(* Logix 5000 project; controller PROJECT2 Emulate 5570 rev 30.12; software revision 30.01; part 3 of 3 *)
(* tags used below, declared in another part *)
   BottleCapped : COUNTER;
   BottleFilled : COUNTER;
   BottlePresentAt4 : TIMER;
   BottlePresentTimer : TIMER;
   CapInsertTimer : TIMER;
   CurrentHeightFilled : DINT;
   CycleTimer : TIMER;
   CycleTimer2 : TIMER;
   Filled : COUNTER;
   filler : BOOL;
   FillerDownTMR : TIMER;
   FillerFilledTMR : TIMER;
   HeightFilled : DINT;
   HEIGHTFILLEDONESHOT : BOOL;
   In : DINT;
   OutPutOneShot : BOOL;
   SIM_BNOP : BOOL;
   SIM_LevelSensor : AOI_SIMAnalogSensor_OnOff;
   SIM_ONS : BOOL;
   SIM_OutfeedSensor : AOI_SIMPartSensor;
   SIM_PowerONPB : BOOL;
   SIM_PPENABLED : BOOL;
   SIM_PTInfeedToStn1 : AOI_SIMPartTravel;
   SIM_PTStn2Fill : AOI_SIMPartTravel;
   SIM_PTStn4ToOutfeed : AOI_SIMPartTravel;
   SIM_PTStnStatus : StationStatus[20];
   SIM_PTWalkingBeam : AOI_SIMPartTravel;
   SIM_SpeedSensor : AOI_SIMAnalogSensor_OnOff;
   SIM_Stn1BottlePresentSensor : AOI_SIMPartSensor;
   SIM_Stn2BottleFilledSensor : AOI_SIMPartSensor;
   SIM_Stn2BottlePresentSensor : AOI_SIMPartSensor;
   SIM_Stn2Filler_Cylinder : AOI_SIM_2PosCyl_RsLwr;
   SIM_Stn2Filler_Fill : AOI_SIM_SimpleValve;
   SIM_Stn3BottlePresentSensor : AOI_SIMPartSensor;
   SIM_Stn3CapInsert : AOI_SIM_2PosCyl_RsLwr;
   SIM_Stn3CapPresentSensor : AOI_SIMPartSensor;
   SIM_Stn4BottlePresentSensor : AOI_SIMPartSensor;
   SIM_Stn4CapRotate : AOI_SIM_Conveyor;
   SIM_Stn4CapRotate_Cylinder : AOI_SIM_2PosCyl_RsLwr;
   SIM_WalkingBeam : AOI_SIM_3PosCyl_ExtRet;
   SIM_WalkingBeamClamp : AOI_SIM_2PosCyl_ExtRet;
   SIM_Zero : DINT;
   St4CycleTime : TIMER;
   station2oneshot : BOOL;
   Station3OneShot : BOOL;
   Station4OneShot : BOOL;
   Station4OneShot2 : BOOL;
   Station4OneShot3 : BOOL;
   TotalCycleTime : REAL;
   TotalFilledHEight : DINT;
   CH0 : ALIAS FOR Local:4:I.Ch0Data;
   CH1 : ALIAS FOR Local:4:I.Ch1Data;
   I2 : ALIAS FOR Local:2:I.Data;
   I31 : ALIAS FOR Ethernet3_PointIO:1:I;
   I32 : ALIAS FOR Ethernet3_PointIO:2:I;
   I33 : ALIAS FOR Ethernet3_PointIO:3:I;
   O3 : ALIAS FOR Local:3:O.Data;
   O34 : ALIAS FOR Ethernet3_PointIO:4:O;
   O35 : ALIAS FOR Ethernet3_PointIO:5:O;
   O36 : ALIAS FOR Ethernet3_PointIO:6:O;
   TP : TouchPanel;
(* MainProgram, continued *)

ROUTINE Filling_R02   (* ladder *)
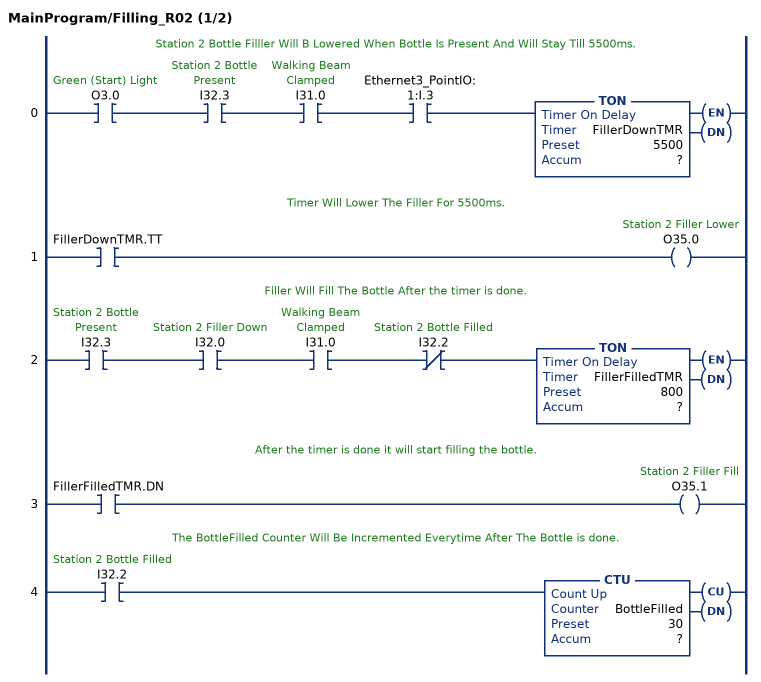
   // Station 2 Bottle Filller Will B Lowered When Bottle Is Present And Will Stay Till 5500ms.
   0: XIC(O3.0)XIC(I32.3)XIC(I31.0)XIC(Ethernet3_PointIO:1:I.3)TON(FillerDownTMR,?,?);
   // Timer Will Lower The Filler For 5500ms.
   1: XIC(FillerDownTMR.TT)OTE(O35.0);
   // Filler Will Fill The Bottle After the timer is done.
   2: XIC(I32.3)XIC(I32.0)XIC(I31.0)XIO(I32.2)TON(FillerFilledTMR,?,?);
   // After the timer is done it will start filling the bottle.
   3: XIC(FillerFilledTMR.DN)OTE(O35.1);
   // The BottleFilled Counter Will Be Incremented Everytime After The Bottle is done.
   4: XIC(I32.2)CTU(BottleFilled,?,?);
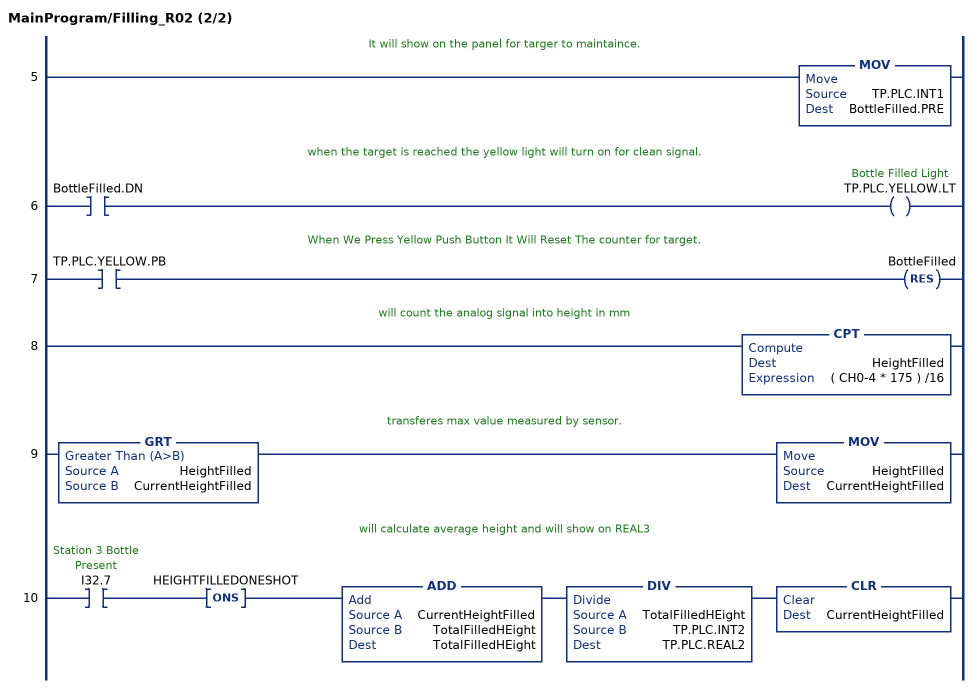
   // It will show on the panel for targer to maintaince.
   5: MOV(TP.PLC.INT1,BottleFilled.PRE);
   // when the target is reached the yellow light will turn on for clean signal.
   6: XIC(BottleFilled.DN)OTE(TP.PLC.YELLOW.LT);
   // When We Press Yellow Push Button It Will Reset The counter for target.
   7: XIC(TP.PLC.YELLOW.PB)RES(BottleFilled);
   // will count the analog signal into height in mm
   8: CPT(HeightFilled,( CH0-4 * 175 ) /16);
   // transferes max value measured by sensor.
   9: GRT(HeightFilled,CurrentHeightFilled)MOV(HeightFilled,CurrentHeightFilled);
   // will calculate average height and will show on REAL3
   10: XIC(I32.7)ONS(HEIGHTFILLEDONESHOT)ADD(CurrentHeightFilled,TotalFilledHEight,TotalFilledHEight)DIV(TotalFilledHEight,TP.PLC.INT2,TP.PLC.REAL2)CLR(CurrentHeightFilled);
END_ROUTINE

ROUTINE MainRoutine   (* ladder *)
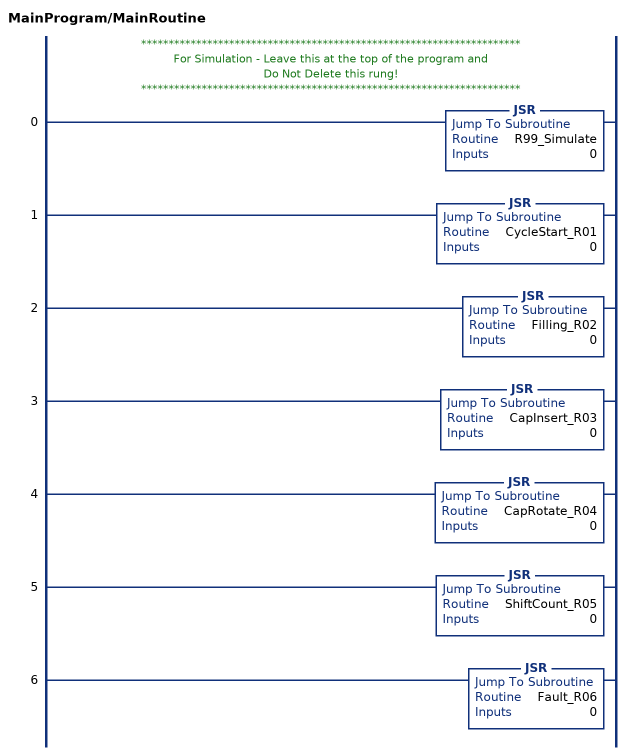
   // *********************************************************************
   // For Simulation - Leave this at the top of the program and
   // Do Not Delete this rung!
   // *********************************************************************
   0: JSR(R99_Simulate,0);
   1: JSR(CycleStart_R01,0);
   2: JSR(Filling_R02,0);
   3: JSR(CapInsert_R03,0);
   4: JSR(CapRotate_R04,0);
   5: JSR(ShiftCount_R05,0);
   6: JSR(Fault_R06,0);
END_ROUTINE

ROUTINE R99_Simulate   (* ladder *)
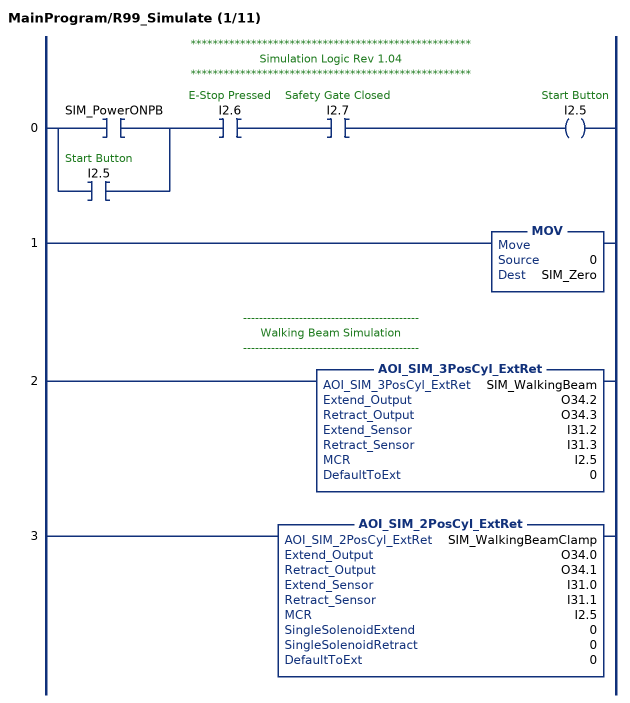
   // ***************************************************
   // Simulation Logic Rev 1.04
   // ***************************************************
   0: [XIC(SIM_PowerONPB) ,XIC(I2.5) ]XIC(I2.6)XIC(I2.7)OTE(I2.5);
   1: MOV(0,SIM_Zero);
   // --------------------------------------------
   // Walking Beam Simulation
   // --------------------------------------------
   2: AOI_SIM_3PosCyl_ExtRet(SIM_WalkingBeam,O34.2,O34.3,I31.2,I31.3,I2.5,0);
   3: AOI_SIM_2PosCyl_ExtRet(SIM_WalkingBeamClamp,O34.0,O34.1,I31.0,I31.1,I2.5,0,0,0);
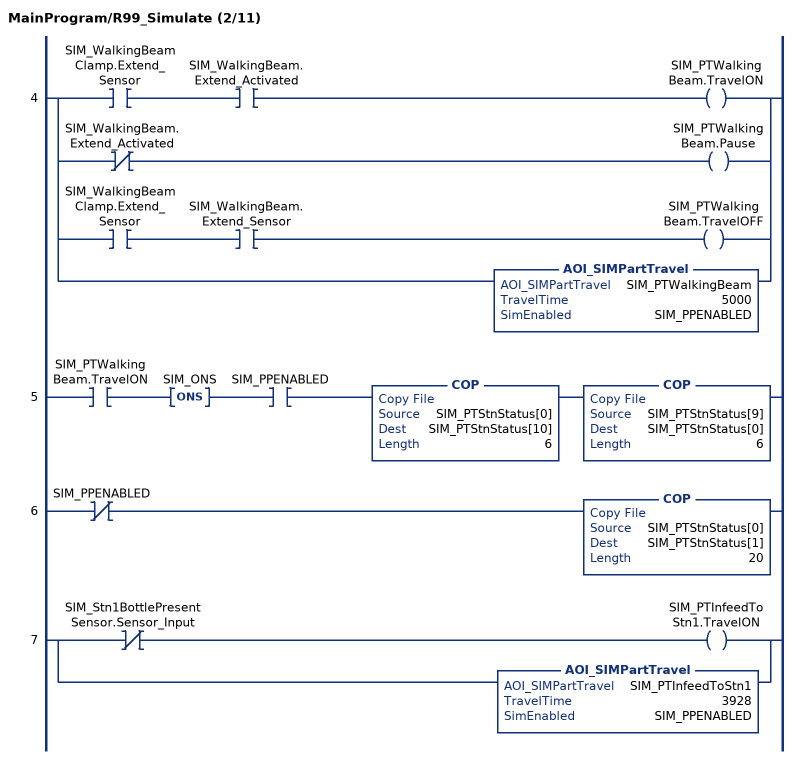
   4: [XIC(SIM_WalkingBeamClamp.Extend_Sensor) XIC(SIM_WalkingBeam.Extend_Activated) OTE(SIM_PTWalkingBeam.TravelON) ,XIO(SIM_WalkingBeam.Extend_Activated) OTE(SIM_PTWalkingBeam.Pause) ,XIC(SIM_WalkingBeamClamp.Extend_Sensor) XIC(SIM_WalkingBeam.Extend_Sensor) OTE(SIM_PTWalkingBeam.TravelOFF) ,AOI_SIMPartTravel(SIM_PTWalkingBeam,5000,SIM_PPENABLED) ];
   5: XIC(SIM_PTWalkingBeam.TravelON)ONS(SIM_ONS)XIC(SIM_PPENABLED)COP(SIM_PTStnStatus[0],SIM_PTStnStatus[10],6)COP(SIM_PTStnStatus[9],SIM_PTStnStatus[0],6);
   6: XIO(SIM_PPENABLED)COP(SIM_PTStnStatus[0],SIM_PTStnStatus[1],20);
   7: [XIO(SIM_Stn1BottlePresentSensor.Sensor_Input) OTE(SIM_PTInfeedToStn1.TravelON) ,AOI_SIMPartTravel(SIM_PTInfeedToStn1,3928,SIM_PPENABLED) ];
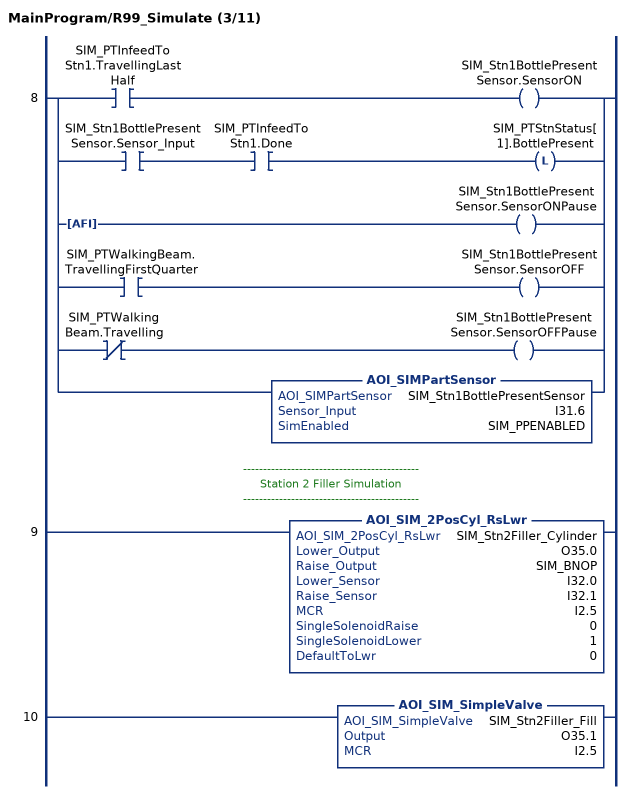
   8: [XIC(SIM_PTInfeedToStn1.TravellingLastHalf) OTE(SIM_Stn1BottlePresentSensor.SensorON) ,XIC(SIM_Stn1BottlePresentSensor.Sensor_Input) XIC(SIM_PTInfeedToStn1.Done) OTL(SIM_PTStnStatus[1].BottlePresent) ,AFI() OTE(SIM_Stn1BottlePresentSensor.SensorONPause) ,XIC(SIM_PTWalkingBeam.TravellingFirstQuarter) OTE(SIM_Stn1BottlePresentSensor.SensorOFF) ,XIO(SIM_PTWalkingBeam.Travelling) OTE(SIM_Stn1BottlePresentSensor.SensorOFFPause) ,AOI_SIMPartSensor(SIM_Stn1BottlePresentSensor,I31.6,SIM_PPENABLED) ];
   // --------------------------------------------
   // Station 2 Filler Simulation
   // --------------------------------------------
   9: AOI_SIM_2PosCyl_RsLwr(SIM_Stn2Filler_Cylinder,O35.0,SIM_BNOP,I32.0,I32.1,I2.5,0,1,0);
   10: AOI_SIM_SimpleValve(SIM_Stn2Filler_Fill,O35.1,I2.5);
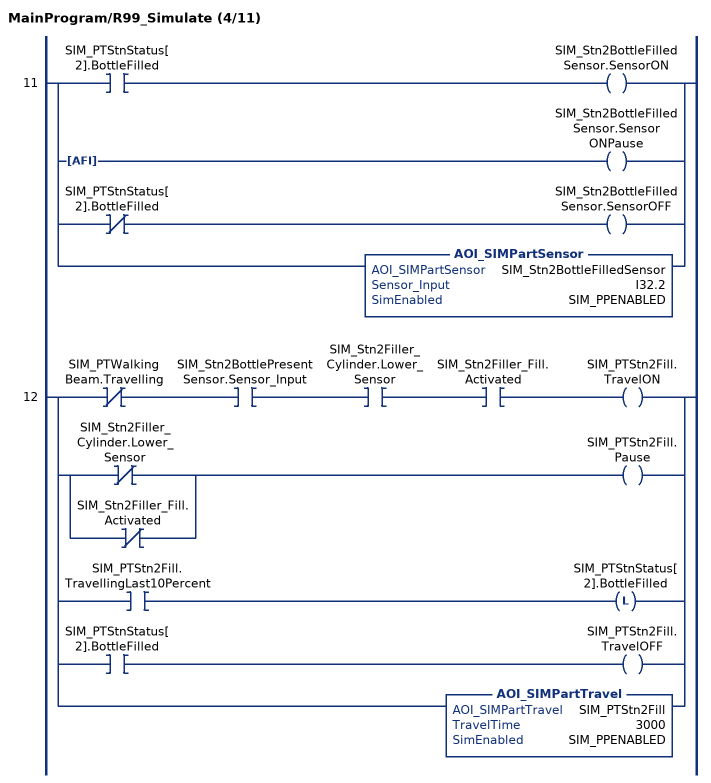
   11: [XIC(SIM_PTStnStatus[2].BottleFilled) OTE(SIM_Stn2BottleFilledSensor.SensorON) ,AFI() OTE(SIM_Stn2BottleFilledSensor.SensorONPause) ,XIO(SIM_PTStnStatus[2].BottleFilled) OTE(SIM_Stn2BottleFilledSensor.SensorOFF) ,AOI_SIMPartSensor(SIM_Stn2BottleFilledSensor,I32.2,SIM_PPENABLED) ];
   12: [XIO(SIM_PTWalkingBeam.Travelling) XIC(SIM_Stn2BottlePresentSensor.Sensor_Input) XIC(SIM_Stn2Filler_Cylinder.Lower_Sensor) XIC(SIM_Stn2Filler_Fill.Activated) OTE(SIM_PTStn2Fill.TravelON) ,[XIO(SIM_Stn2Filler_Cylinder.Lower_Sensor) ,XIO(SIM_Stn2Filler_Fill.Activated) ] OTE(SIM_PTStn2Fill.Pause) ,XIC(SIM_PTStn2Fill.TravellingLast10Percent) OTL(SIM_PTStnStatus[2].BottleFilled) ,XIC(SIM_PTStnStatus[2].BottleFilled) OTE(SIM_PTStn2Fill.TravelOFF) ,AOI_SIMPartTravel(SIM_PTStn2Fill,3000,SIM_PPENABLED) ];
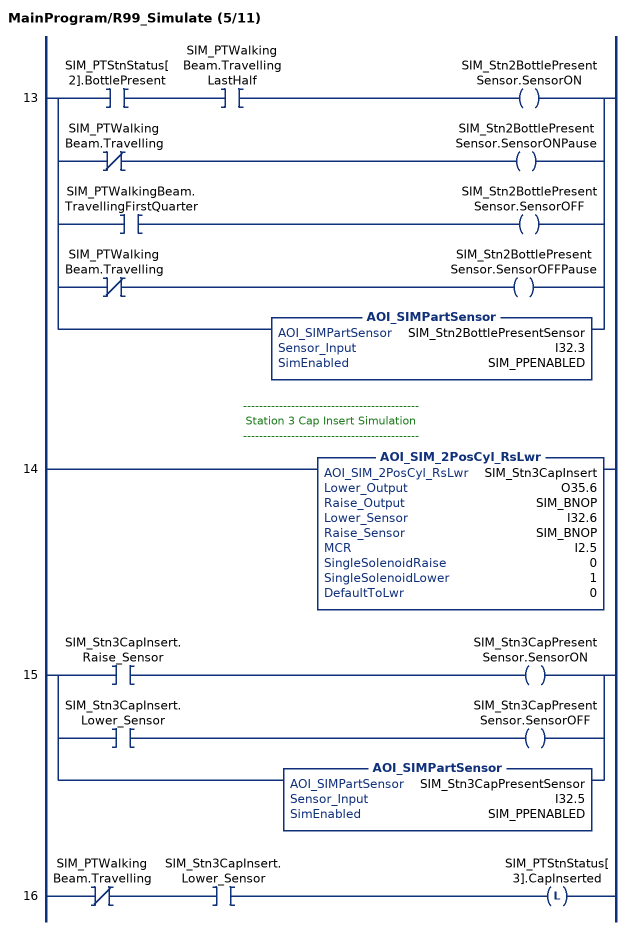
   13: [XIC(SIM_PTStnStatus[2].BottlePresent) XIC(SIM_PTWalkingBeam.TravellingLastHalf) OTE(SIM_Stn2BottlePresentSensor.SensorON) ,XIO(SIM_PTWalkingBeam.Travelling) OTE(SIM_Stn2BottlePresentSensor.SensorONPause) ,XIC(SIM_PTWalkingBeam.TravellingFirstQuarter) OTE(SIM_Stn2BottlePresentSensor.SensorOFF) ,XIO(SIM_PTWalkingBeam.Travelling) OTE(SIM_Stn2BottlePresentSensor.SensorOFFPause) ,AOI_SIMPartSensor(SIM_Stn2BottlePresentSensor,I32.3,SIM_PPENABLED) ];
   // --------------------------------------------
   // Station 3 Cap Insert Simulation
   // --------------------------------------------
   14: AOI_SIM_2PosCyl_RsLwr(SIM_Stn3CapInsert,O35.6,SIM_BNOP,I32.6,SIM_BNOP,I2.5,0,1,0);
   15: [XIC(SIM_Stn3CapInsert.Raise_Sensor) OTE(SIM_Stn3CapPresentSensor.SensorON) ,XIC(SIM_Stn3CapInsert.Lower_Sensor) OTE(SIM_Stn3CapPresentSensor.SensorOFF) ,AOI_SIMPartSensor(SIM_Stn3CapPresentSensor,I32.5,SIM_PPENABLED) ];
   16: XIO(SIM_PTWalkingBeam.Travelling)XIC(SIM_Stn3CapInsert.Lower_Sensor)OTL(SIM_PTStnStatus[3].CapInserted);
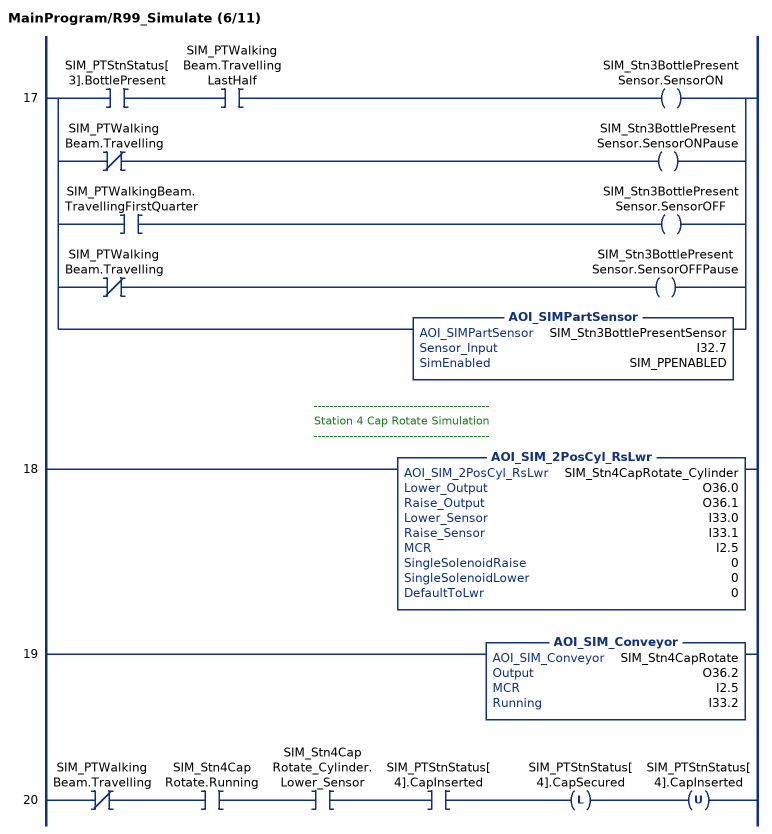
   17: [XIC(SIM_PTStnStatus[3].BottlePresent) XIC(SIM_PTWalkingBeam.TravellingLastHalf) OTE(SIM_Stn3BottlePresentSensor.SensorON) ,XIO(SIM_PTWalkingBeam.Travelling) OTE(SIM_Stn3BottlePresentSensor.SensorONPause) ,XIC(SIM_PTWalkingBeam.TravellingFirstQuarter) OTE(SIM_Stn3BottlePresentSensor.SensorOFF) ,XIO(SIM_PTWalkingBeam.Travelling) OTE(SIM_Stn3BottlePresentSensor.SensorOFFPause) ,AOI_SIMPartSensor(SIM_Stn3BottlePresentSensor,I32.7,SIM_PPENABLED) ];
   // --------------------------------------------
   // Station 4 Cap Rotate Simulation
   // --------------------------------------------
   18: AOI_SIM_2PosCyl_RsLwr(SIM_Stn4CapRotate_Cylinder,O36.0,O36.1,I33.0,I33.1,I2.5,0,0,0);
   19: AOI_SIM_Conveyor(SIM_Stn4CapRotate,O36.2,I2.5,I33.2);
   20: XIO(SIM_PTWalkingBeam.Travelling)XIC(SIM_Stn4CapRotate.Running)XIC(SIM_Stn4CapRotate_Cylinder.Lower_Sensor)XIC(SIM_PTStnStatus[4].CapInserted)OTL(SIM_PTStnStatus[4].CapSecured)OTU(SIM_PTStnStatus[4].CapInserted);
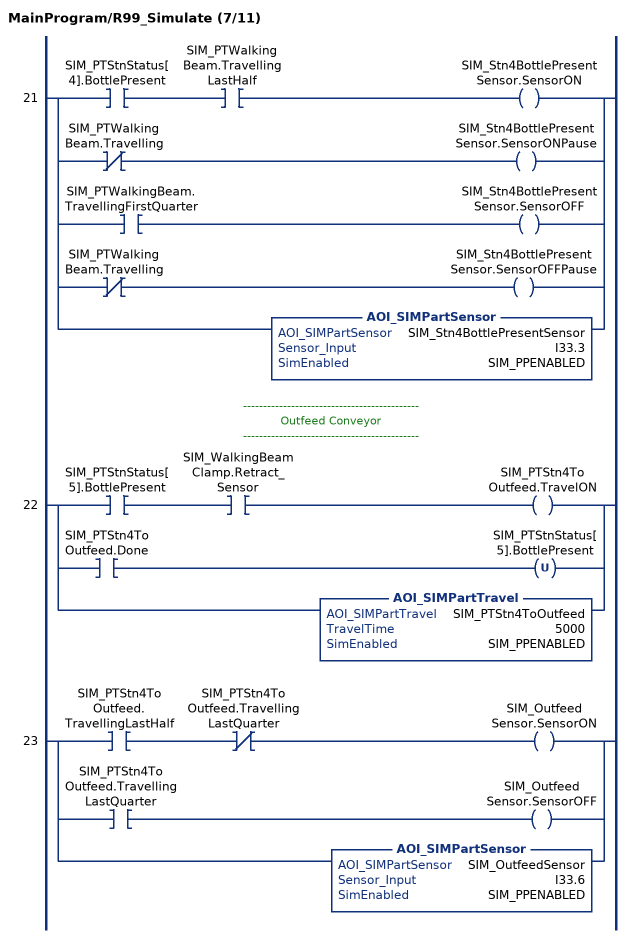
   21: [XIC(SIM_PTStnStatus[4].BottlePresent) XIC(SIM_PTWalkingBeam.TravellingLastHalf) OTE(SIM_Stn4BottlePresentSensor.SensorON) ,XIO(SIM_PTWalkingBeam.Travelling) OTE(SIM_Stn4BottlePresentSensor.SensorONPause) ,XIC(SIM_PTWalkingBeam.TravellingFirstQuarter) OTE(SIM_Stn4BottlePresentSensor.SensorOFF) ,XIO(SIM_PTWalkingBeam.Travelling) OTE(SIM_Stn4BottlePresentSensor.SensorOFFPause) ,AOI_SIMPartSensor(SIM_Stn4BottlePresentSensor,I33.3,SIM_PPENABLED) ];
   // --------------------------------------------
   // Outfeed Conveyor
   // --------------------------------------------
   22: [XIC(SIM_PTStnStatus[5].BottlePresent) XIC(SIM_WalkingBeamClamp.Retract_Sensor) OTE(SIM_PTStn4ToOutfeed.TravelON) ,XIC(SIM_PTStn4ToOutfeed.Done) OTU(SIM_PTStnStatus[5].BottlePresent) ,AOI_SIMPartTravel(SIM_PTStn4ToOutfeed,5000,SIM_PPENABLED) ];
   23: [XIC(SIM_PTStn4ToOutfeed.TravellingLastHalf) XIO(SIM_PTStn4ToOutfeed.TravellingLastQuarter) OTE(SIM_OutfeedSensor.SensorON) ,XIC(SIM_PTStn4ToOutfeed.TravellingLastQuarter) OTE(SIM_OutfeedSensor.SensorOFF) ,AOI_SIMPartSensor(SIM_OutfeedSensor,I33.6,SIM_PPENABLED) ];
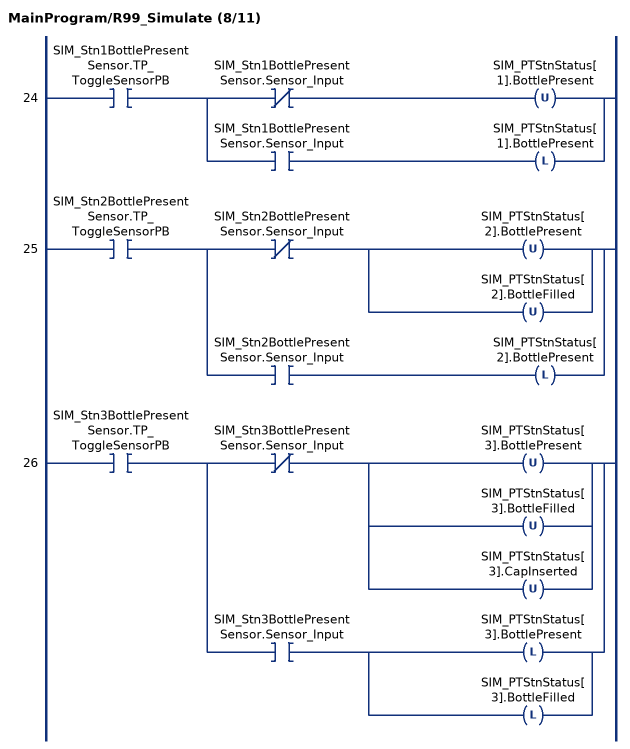
   24: XIC(SIM_Stn1BottlePresentSensor.TP_ToggleSensorPB)[XIO(SIM_Stn1BottlePresentSensor.Sensor_Input) OTU(SIM_PTStnStatus[1].BottlePresent) ,XIC(SIM_Stn1BottlePresentSensor.Sensor_Input) OTL(SIM_PTStnStatus[1].BottlePresent) ];
   25: XIC(SIM_Stn2BottlePresentSensor.TP_ToggleSensorPB)[XIO(SIM_Stn2BottlePresentSensor.Sensor_Input) [OTU(SIM_PTStnStatus[2].BottlePresent) ,OTU(SIM_PTStnStatus[2].BottleFilled) ] ,XIC(SIM_Stn2BottlePresentSensor.Sensor_Input) OTL(SIM_PTStnStatus[2].BottlePresent) ];
   26: XIC(SIM_Stn3BottlePresentSensor.TP_ToggleSensorPB)[XIO(SIM_Stn3BottlePresentSensor.Sensor_Input) [OTU(SIM_PTStnStatus[3].BottlePresent) ,OTU(SIM_PTStnStatus[3].BottleFilled) ,OTU(SIM_PTStnStatus[3].CapInserted) ] ,XIC(SIM_Stn3BottlePresentSensor.Sensor_Input) [OTL(SIM_PTStnStatus[3].BottlePresent) ,OTL(SIM_PTStnStatus[3].BottleFilled) ] ];
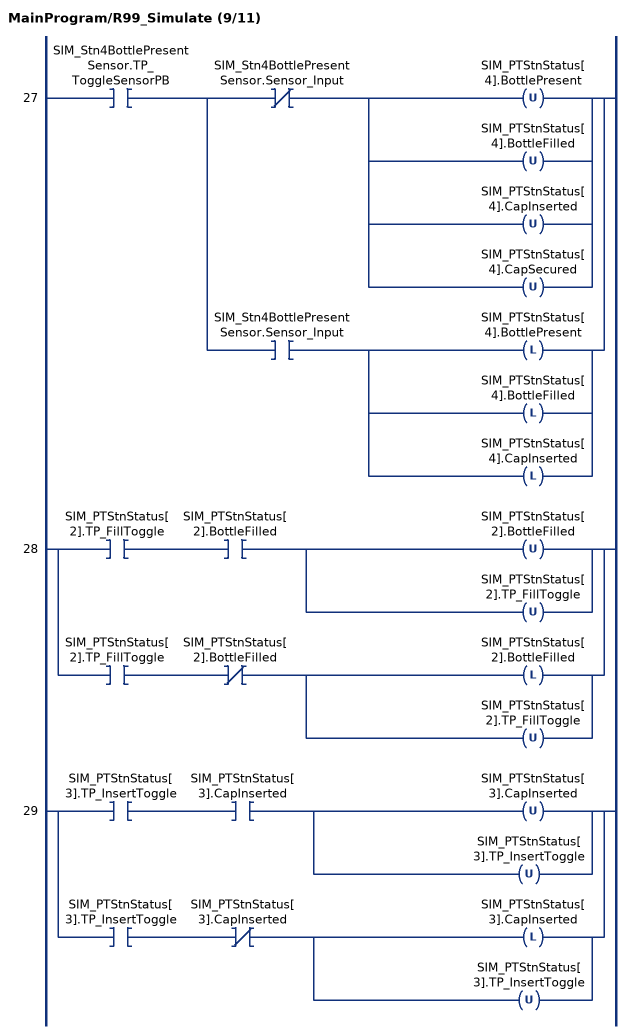
   27: XIC(SIM_Stn4BottlePresentSensor.TP_ToggleSensorPB)[XIO(SIM_Stn4BottlePresentSensor.Sensor_Input) [OTU(SIM_PTStnStatus[4].BottlePresent) ,OTU(SIM_PTStnStatus[4].BottleFilled) ,OTU(SIM_PTStnStatus[4].CapInserted) ,OTU(SIM_PTStnStatus[4].CapSecured) ] ,XIC(SIM_Stn4BottlePresentSensor.Sensor_Input) [OTL(SIM_PTStnStatus[4].BottlePresent) ,OTL(SIM_PTStnStatus[4].BottleFilled) ,OTL(SIM_PTStnStatus[4].CapInserted) ] ];
   28: [XIC(SIM_PTStnStatus[2].TP_FillToggle) XIC(SIM_PTStnStatus[2].BottleFilled) [OTU(SIM_PTStnStatus[2].BottleFilled) ,OTU(SIM_PTStnStatus[2].TP_FillToggle) ] ,XIC(SIM_PTStnStatus[2].TP_FillToggle) XIO(SIM_PTStnStatus[2].BottleFilled) [OTL(SIM_PTStnStatus[2].BottleFilled) ,OTU(SIM_PTStnStatus[2].TP_FillToggle) ] ];
   29: [XIC(SIM_PTStnStatus[3].TP_InsertToggle) XIC(SIM_PTStnStatus[3].CapInserted) [OTU(SIM_PTStnStatus[3].CapInserted) ,OTU(SIM_PTStnStatus[3].TP_InsertToggle) ] ,XIC(SIM_PTStnStatus[3].TP_InsertToggle) XIO(SIM_PTStnStatus[3].CapInserted) [OTL(SIM_PTStnStatus[3].CapInserted) ,OTU(SIM_PTStnStatus[3].TP_InsertToggle) ] ];
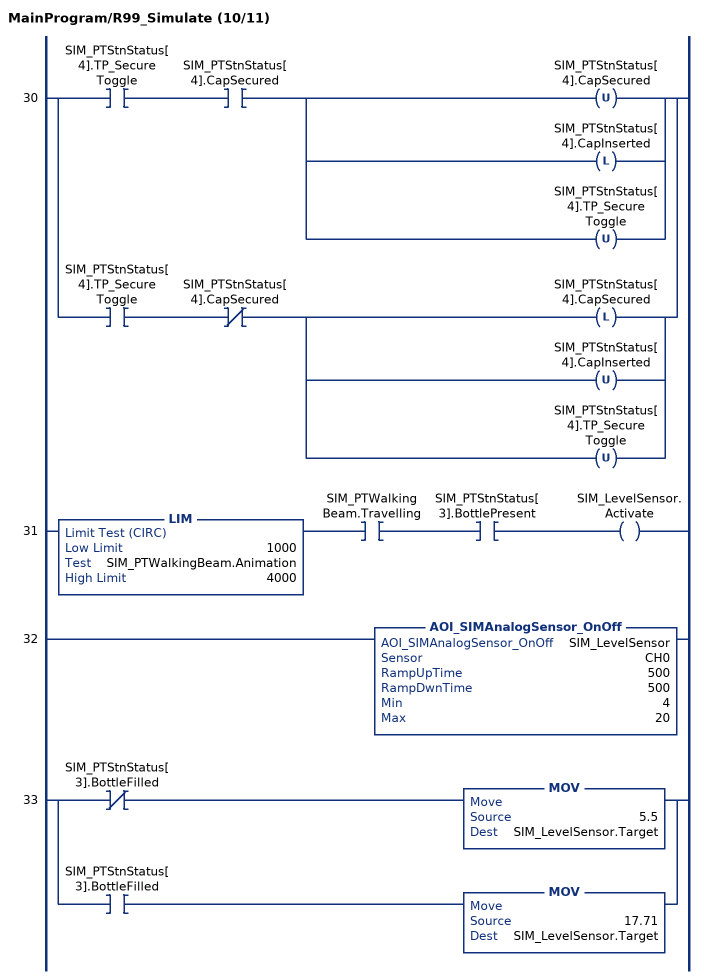
   30: [XIC(SIM_PTStnStatus[4].TP_SecureToggle) XIC(SIM_PTStnStatus[4].CapSecured) [OTU(SIM_PTStnStatus[4].CapSecured) ,OTL(SIM_PTStnStatus[4].CapInserted) ,OTU(SIM_PTStnStatus[4].TP_SecureToggle) ] ,XIC(SIM_PTStnStatus[4].TP_SecureToggle) XIO(SIM_PTStnStatus[4].CapSecured) [OTL(SIM_PTStnStatus[4].CapSecured) ,OTU(SIM_PTStnStatus[4].CapInserted) ,OTU(SIM_PTStnStatus[4].TP_SecureToggle) ] ];
   31: LIM(1000,SIM_PTWalkingBeam.Animation,4000)XIC(SIM_PTWalkingBeam.Travelling)XIC(SIM_PTStnStatus[3].BottlePresent)OTE(SIM_LevelSensor.Activate);
   32: AOI_SIMAnalogSensor_OnOff(SIM_LevelSensor,CH0,500,500,4,20);
   33: [XIO(SIM_PTStnStatus[3].BottleFilled) MOV(5.5,SIM_LevelSensor.Target) ,XIC(SIM_PTStnStatus[3].BottleFilled) MOV(17.71,SIM_LevelSensor.Target) ];
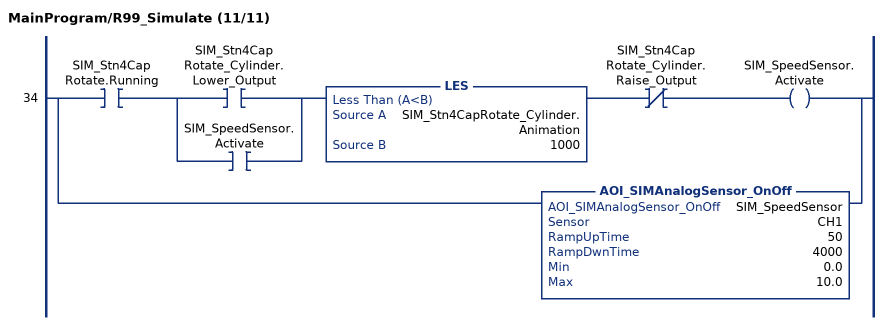
   34: [XIC(SIM_Stn4CapRotate.Running) [XIC(SIM_Stn4CapRotate_Cylinder.Lower_Output) ,XIC(SIM_SpeedSensor.Activate) ] LES(SIM_Stn4CapRotate_Cylinder.Animation,1000) XIO(SIM_Stn4CapRotate_Cylinder.Raise_Output) OTE(SIM_SpeedSensor.Activate) ,AOI_SIMAnalogSensor_OnOff(SIM_SpeedSensor,CH1,50,4000,0.0,10.0) ];
END_ROUTINE

ROUTINE ShiftCount_R05   (* ladder *)
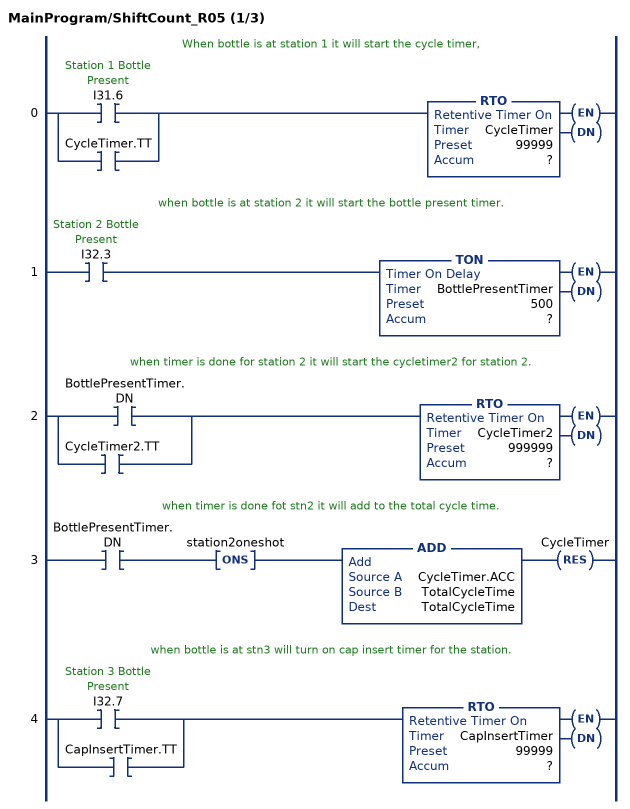
   // When bottle is at station 1 it will start the cycle timer,
   0: [XIC(I31.6) ,XIC(CycleTimer.TT) ]RTO(CycleTimer,?,?);
   // when bottle is at station 2 it will start the bottle present timer.
   1: XIC(I32.3)TON(BottlePresentTimer,?,?);
   // when timer is done for station 2 it will start the cycletimer2 for station 2.
   2: [XIC(BottlePresentTimer.DN) ,XIC(CycleTimer2.TT) ]RTO(CycleTimer2,?,?);
   // when timer is done fot stn2 it will add to the total cycle time.
   3: XIC(BottlePresentTimer.DN)ONS(station2oneshot)ADD(CycleTimer.ACC,TotalCycleTime,TotalCycleTime)RES(CycleTimer);
   // when bottle is at stn3 will turn on cap insert timer for the station.
   4: [XIC(I32.7) ,XIC(CapInsertTimer.TT) ]RTO(CapInsertTimer,?,?);
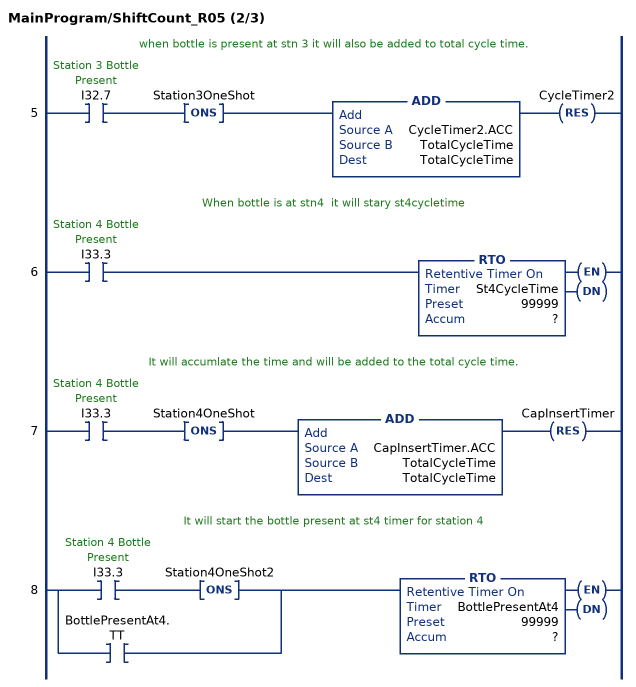
   // when bottle is present at stn 3 it will also be added to total cycle time.
   5: XIC(I32.7)ONS(Station3OneShot)ADD(CycleTimer2.ACC,TotalCycleTime,TotalCycleTime)RES(CycleTimer2);
   // When bottle is at stn4  it will stary st4cycletime
   6: XIC(I33.3)RTO(St4CycleTime,?,?);
   // It will accumlate the time and will be added to the total cycle time.
   7: XIC(I33.3)ONS(Station4OneShot)ADD(CapInsertTimer.ACC,TotalCycleTime,TotalCycleTime)RES(CapInsertTimer);
   // It will start the bottle present at st4 timer for station 4
   8: [XIC(I33.3) ONS(Station4OneShot2) ,XIC(BottlePresentAt4.TT) ]RTO(BottlePresentAt4,?,?);
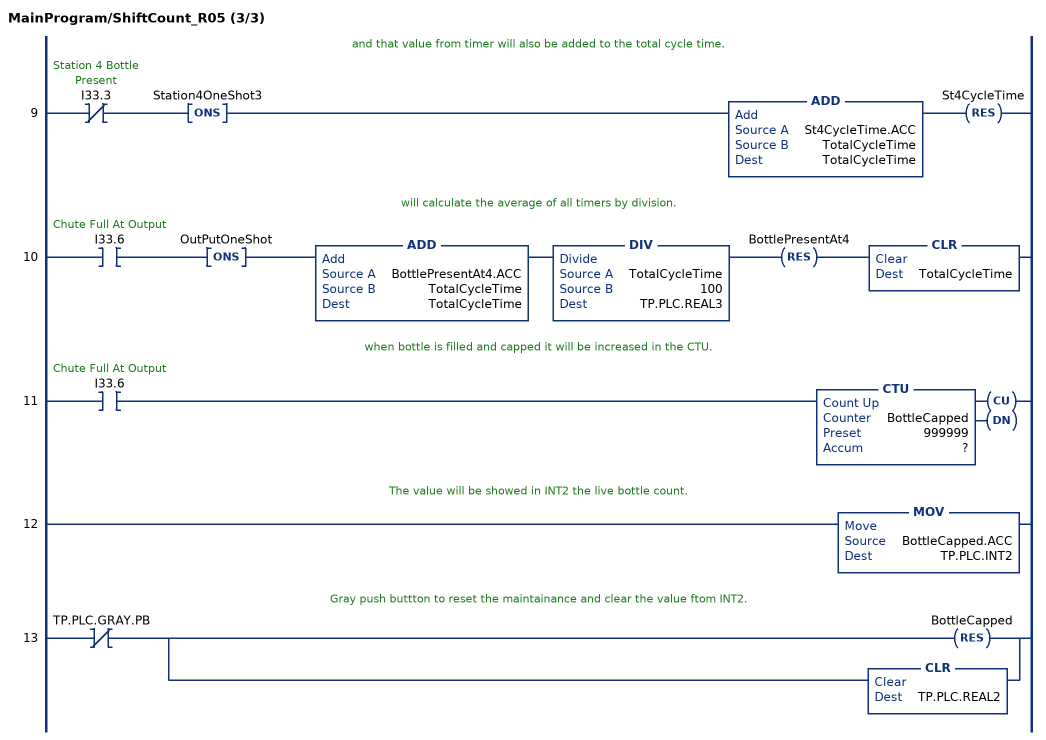
   // and that value from timer will also be added to the total cycle time.
   9: XIO(I33.3)ONS(Station4OneShot3)ADD(St4CycleTime.ACC,TotalCycleTime,TotalCycleTime)RES(St4CycleTime);
   // will calculate the average of all timers by division.
   10: XIC(I33.6)ONS(OutPutOneShot)ADD(BottlePresentAt4.ACC,TotalCycleTime,TotalCycleTime)DIV(TotalCycleTime,100,TP.PLC.REAL3)RES(BottlePresentAt4)CLR(TotalCycleTime);
   // when bottle is filled and capped it will be increased in the CTU.
   11: XIC(I33.6)CTU(BottleCapped,?,?);
   // The value will be showed in INT2 the live bottle count.
   12: MOV(BottleCapped.ACC,TP.PLC.INT2);
   // Gray push buttton to reset the maintainance and clear the value ftom INT2.
   13: XIO(TP.PLC.GRAY.PB)[RES(BottleCapped) ,CLR(TP.PLC.REAL2) ];
END_ROUTINE
END_PROGRAM
